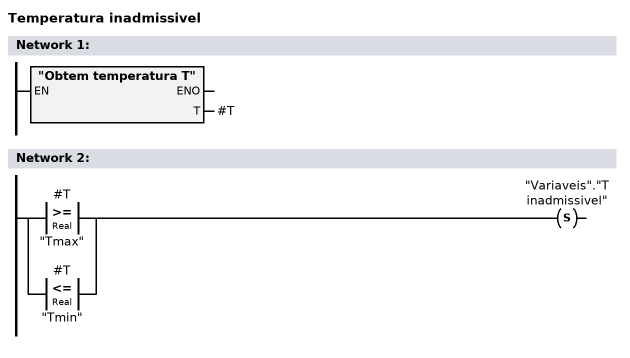
   RUNG wire#powerrail
      "Obtem temperatura T"(T => #T)
   END_RUNG
   // the same network as SCL:
   "Obtem temperatura T"(T => #T);
END_REGION

REGION Network 2
   RUNG wire#powerrail
      { S7_Templates := "SrcType := Real" } GE_Contact(in1 := #T, in2 := "Tmax")
      wire#w1
      S_Coil( "Variaveis"."T inadmissivel" )
   END_RUNG
   RUNG wire#powerrail
      { S7_Templates := "SrcType := Real" } LE_Contact(in1 := #T, in2 := "Tmin")
   END_RUNG wire#w1
   // the same network as SCL:
   IF (#T >= "Tmax") OR (#T <= "Tmin") THEN "Variaveis"."T inadmissivel" := TRUE; END_IF;
END_REGION
END_FUNCTION

FUNCTION "Pisca LED3" : Void   // FC45, LAD
{ S7_Optimized_Access := 'TRUE' }
VERSION : 0.1
   VAR_TEMP   // added for the SCL form of the ladder/FBD networks
      _w1 : Bool;
   END_VAR
BEGIN

REGION Network 1: LED que avisa sobre a pressão no tanque separador
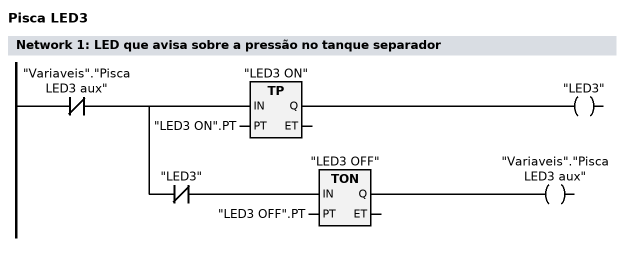
   #_w1 := NOT "Variaveis"."Pisca LED3 aux";
   "LED3 ON".TP(IN := #_w1, PT := "LED3 ON".PT);
   "LED3" := "LED3 ON".Q;
   "LED3 OFF".TON(IN := #_w1 AND NOT "LED3", PT := "LED3 OFF".PT);
   "Variaveis"."Pisca LED3 aux" := "LED3 OFF".Q;
END_REGION
END_FUNCTION

ORGANIZATION_BLOCK "Main"   // OB1, LAD, ProgramCycle
TITLE = "Main Program Sweep (Cycle)"
{ S7_Optimized_Access := 'TRUE' }
VERSION : 0.1
   VAR_INPUT
      Initial_Call : Bool;   // Initial call of this OB
      Remanence : Bool;   // =True, if remanent data are available
   END_VAR
BEGIN

REGION Network 1: LED que avisa sobre a pressão no tanque separador
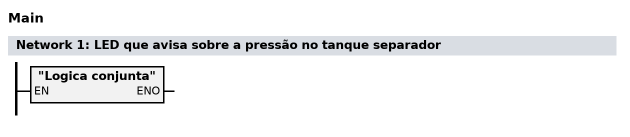
   RUNG wire#powerrail
      "Logica conjunta"()
   END_RUNG
   // the same network as SCL:
   "Logica conjunta"();
END_REGION
END_ORGANIZATION_BLOCK